FUNCTION_BLOCK DoorOpenBasketTransfer
VAR_INPUT

	bMainOnOff:BOOL;
	bDownPost:BOOL;
	bHookPost:BOOL;
	bBasketComfirm:BOOL;

	bNextDownPost:BOOL;
	bNextUnHookPost:BOOL;



END_VAR
VAR_OUTPUT
	bBasketTransfer:BOOL;

END_VAR
VAR
	BasketTransferComplete: BOOL;
END_VAR

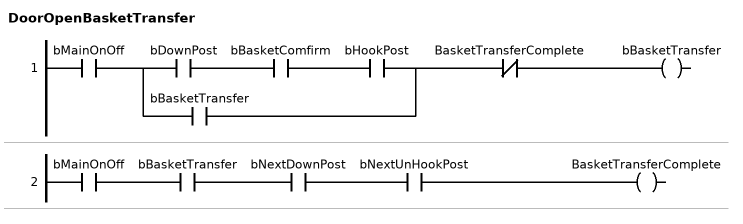
// NETWORK 1
bBasketTransfer := (bMainOnOff AND (bDownPost AND bBasketComfirm AND bHookPost OR bBasketTransfer)) AND NOT BasketTransferComplete;

// NETWORK 2
BasketTransferComplete := bMainOnOff AND bBasketTransfer AND bNextDownPost AND bNextUnHookPost;

END_FUNCTION_BLOCK

(* stored: Version 1.1.0.1, ProductVersion 3.1.4024.12
   POU DoorOpenBasketTransfer: Id {8dbc184a-185f-460a-8cb8-b2212a6d619c}, SpecialFunc None *)
